(* IEC 61131-3 sources: repolevel_ST_code_completion/output/0127完整版本_带planner/repoeval_assembly-station/readful_result_before_fix, 1 file *)

(* ---- PNP_MACHINE.st ---- *)
FUNCTION_BLOCK PUBLIC PNP_MACHINE
VAR_INPUT
	BaseClamped: BOOL;
	LidClamped: BOOL;
	Reset: BOOL := FALSE;
END_VAR

VAR_OUTPUT
	LidPicked: BOOL := FALSE;
	LidPlaced: BOOL := FALSE;
END_VAR
VAR
	FB_ItemDetect : R_TRIG;
	FB_MovingZ: F_TRIG;
	FB_MovingX : F_TRIG;

	_pickerMoved: BOOL := FALSE;
	_movePicker: BOOL := FALSE;
	_moveArm: BOOL := FALSE;
	_armMoved : BOOL := FALSE;
	_grabItem: BOOL := FALSE;
	_itemDetected: BOOL := FALSE;
	_gripperAtLid: BOOL := FALSE;
	_gripperAtBase: BOOL := FALSE;
END_VAR

FB_MovingZ(CLK := FIO.FIO_iMovingZ);
FB_MovingX(CLK := FIO.FIO_iMovingX);
FB_ItemDetect(CLK := FIO.FIO_iItemDetected);

FIO.FIO_oMoveZ := _movePicker;
FIO.FIO_oGrab := _grabItem;
FIO.FIO_oMoveX := _moveArm;

IF Reset THEN
	_pickerMoved := FALSE;
	_movePicker := FALSE;
	_grabItem := FALSE;
	_moveArm := FALSE;
	_armMoved := FALSE;
	LidPicked := FALSE;
	LidPlaced := FALSE;
	_itemDetected := FALSE;
	_gripperAtLid := FALSE;
	_gripperAtBase := FALSE;
	RETURN;
END_IF;

IF BaseClamped AND LidClamped THEN
	IF NOT LidPicked THEN
		_gripperAtLid := TRUE;
		_grabItem := TRUE;
		_movePicker := TRUE;
		IF FB_MovingZ.Q THEN
			_pickerMoved := TRUE;
			_grabItem := FALSE;
			LidPicked := TRUE;
		END_IF;
	END_IF;

	IF LidPicked AND NOT LidPlaced THEN
		_gripperAtLid := FALSE;
		_gripperAtBase := TRUE;
		_moveArm := TRUE;
		IF FB_MovingX.Q THEN
			_armMoved := TRUE;
			_moveArm := FALSE;
			_grabItem := TRUE;
			IF FB_MovingZ.Q THEN
				LidPlaced := TRUE;
				_grabItem := FALSE;
			END_IF;
		END_IF;
	END_IF;

	IF LidPlaced THEN
		_pickerMoved := FALSE;
		_armMoved := FALSE;
		LidPicked := FALSE;
		LidPlaced := FALSE;
		_gripperAtBase := FALSE;
	END_IF;
END_IF;
END_FUNCTION_BLOCK
